// TIA Portal project "timer" (V14)

(* hardware
DEVICE "S7-1200 station_1"  S7-1200 Station
   slot 0: "Rack_0"  S7-1200 Rack  Rack  V1.0
   slot 1: "PLC_1"  CPU 1212C DC/DC/DC  6ES7 212-1AE40-0XB0  V4.2
*)

// ===== PLC "PLC_1"  CPU 1212C DC/DC/DC =====

VAR_GLOBAL   // PLC tag table "Default tag table"
   ""start1"" AT %I0.0 : Bool;
   ""stop1"" AT %I0.1 : Bool;
   ""Tag_3"" AT %I0.2 : Bool;
   ""Tag_4"" AT %I0.3 : Bool;
   ""motor1"" AT %Q0.0 : Bool;
   ""motor2"" AT %Q0.1 : Bool;
END_VAR